// TIA Portal project "2022.06.11_液位控制" (V17)

(* hardware
DEVICE "S7-1200 station_1"  S7-1200 Station
   slot 0: "Rack_0"  S7-1200 Rack  Rack  V1.0
   slot 1: "PLC_1"  CPU 1212C DC/DC/DC  6ES7 212-1AE40-0XB0  V4.5
   slot 2: "AI 4x13BIT/AQ 2x14BIT_1"  SM 1234 AI4/AQ2  6ES7 234-4HE30-0XB0  V1.0
*)

// ===== PLC "PLC_1"  CPU 1212C DC/DC/DC =====

VAR_GLOBAL   // PLC tag table "默认变量表"
   "液位测量" AT %IW96 : Word;
   "百分比" AT %MD40 : DWord;
   "模拟量输出通道" AT %MD44 : UDInt;
   "所需频率(1)" AT %MD0 : Real;
   "压力2模拟输入通道" AT %IW100 : Int;
   "液位" AT %MD4 : Real;
   "频率" AT %MD8 : Real;
   "Tag_2" AT %MD12 : Real;
   "模拟量输出" AT %QW96 : Int;
   "设定液位值" AT %MD20 : Real;
   "实际液位值" AT %MD24 : Real;
END_VAR

ORGANIZATION_BLOCK "Main"   // OB1, LAD, ProgramCycle
TITLE = "Main Program Sweep (Cycle)"
{ S7_Optimized_Access := 'TRUE' }
VERSION : 0.1
   VAR_INPUT
      Initial_Call : Bool;   // Initial call of this OB
      Remanence : Bool;   // =True, if remanent data are available
   END_VAR
BEGIN

REGION Network 1
   // 测试液位传感器，模拟量输入
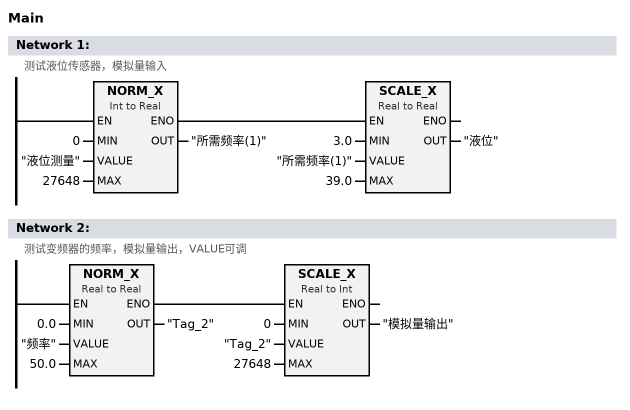
   RUNG wire#powerrail
      { S7_Templates := "[SrcType := Int, DestType := Real]" } Normalize(min := 0, value := "液位测量", max := 27648, out => "所需频率(1)")
      { S7_Templates := "[SrcType := Real, DestType := Real]" } Scale(min := 3.0, value := "所需频率(1)", max := 39.0, out => "液位")
   END_RUNG
   // the same network as SCL:
   "所需频率(1)" := NORM_X(MIN := 0, VALUE := "液位测量", MAX := 27648);
   "液位" := SCALE_X(MIN := 3.0, VALUE := "所需频率(1)", MAX := 39.0);
END_REGION

REGION Network 2
   // 测试变频器的频率，模拟量输出，VALUE可调
   RUNG wire#powerrail
      { S7_Templates := "[SrcType := Real, DestType := Real]" } Normalize(min := 0.0, value := "频率", max := 50.0, out => "Tag_2")
      { S7_Templates := "[SrcType := Real, DestType := Int]" } Scale(min := 0, value := "Tag_2", max := 27648, out => "模拟量输出")
   END_RUNG
   // the same network as SCL:
   "Tag_2" := NORM_X(MIN := 0.0, VALUE := "频率", MAX := 50.0);
   "模拟量输出" := SCALE_X(MIN := 0, VALUE := "Tag_2", MAX := 27648);
END_REGION
END_ORGANIZATION_BLOCK

ORGANIZATION_BLOCK "Cyclic interrupt"   // OB30, LAD, CyclicInterrupt
{ S7_Optimized_Access := 'TRUE' }
VERSION : 0.1
   VAR_INPUT
      Initial_Call : Bool;   // Initial call of this OB
      Event_Count : Int;   // Events discarded
   END_VAR
BEGIN

REGION Network 1
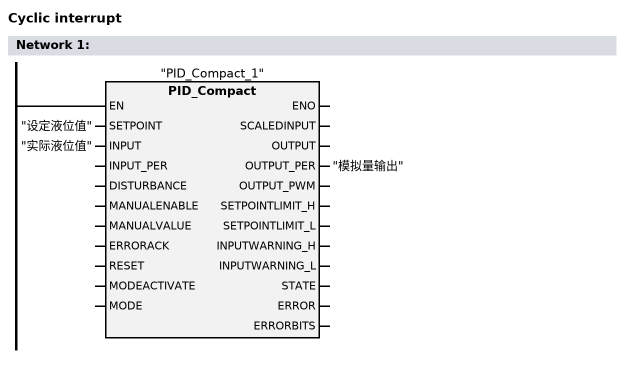
   "PID_Compact_1"(Setpoint := "设定液位值", Input := "实际液位值", Output_PER => "模拟量输出");   // PID_Compact
END_REGION
END_ORGANIZATION_BLOCK